PROGRAM P_SafetyErrors
VAR
END_VAR

IF GVL_Safe_IO.bCom_Error OR 
		GVL_Safe_IO.bFB_Error OR
		GVL_Safe_IO.bOut_Error  THEN
	GVL_PLC.bSafetyError := TRUE;
END_IF





IF GVL_Safe_IO.bAck_Error THEN
	GVL_PLC.bSafetyError := FALSE;
END_IF

END_PROGRAM

(* stored: Version 1.1.0.1, ProductVersion 3.1.4022.3
   POU P_SafetyErrors: Id {4d8975fb-66fe-4347-ac0b-2c21e0904f31}, SpecialFunc None *)
